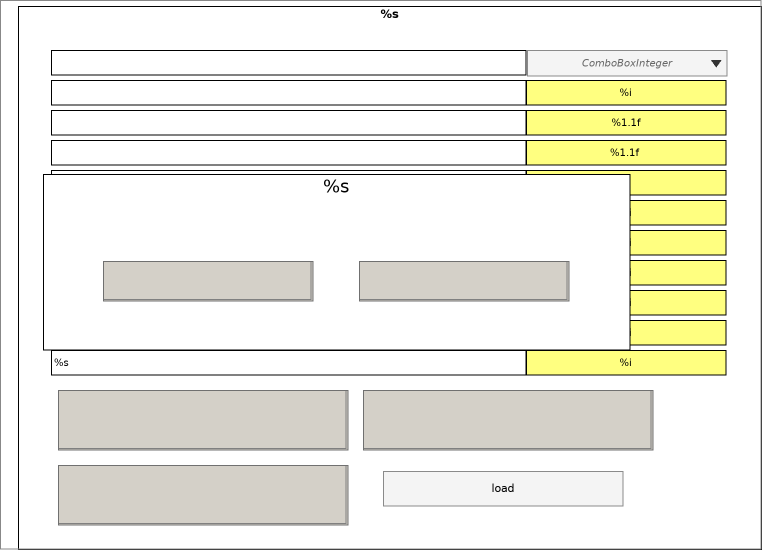
VISUALIZATION VISU_REGENERATION  // 762x550
VAR_IN_OUT
	COM: BLOCK_RS232_ONBOARD_V4;
END_VAR
    RoundedRectangle (18,6 744x544), "%s", text list: 'TextList_CryoPump', text index: 98
    Rectangle (51,50 475x25), text list: 'TextList_CryoPump', text index: 45
    Rectangle (526,140 200x25), "%1.1f", text variable: COM.PRM_PumpRestartDelay, input disabled if: NOT Global_Variables.PRG_USER.ACTU_USER.CONF_MACHINE
        OnMouseClick: write COM.PRM_PumpRestartDelay via Edit
    Rectangle (51,110 475x25), text list: 'TextList_CryoPump', text index: 57
    Rectangle (51,140 475x25), text list: 'TextList_CryoPump', text index: 11
    Rectangle (51,170 475x25), text list: 'TextList_CryoPump', text index: 10
    Rectangle (51,200 475x25), text list: 'TextList_CryoPump', text index: 12
    Rectangle (51,230 475x25), text list: 'TextList_CryoPump', text index: 13
    Rectangle (51,260 475x25), text list: 'TextList_CryoPump', text index: 30
    Progressbar (383,471 240x35), "load", variable: COM.iCounter_Regen_lecture, invisible if: not(COM.VAR_Mem_CO_Lecture)
    Rectangle (526,110 200x25), "%1.1f", text variable: COM.PRM_PumpStartDelay, input disabled if: NOT Global_Variables.PRG_USER.ACTU_USER.CONF_MACHINE
        OnMouseClick: write COM.PRM_PumpStartDelay via Edit
    ComboBoxInteger (527,50 200x26), variable: COM.ID_COMBOBOX, input disabled if: NOT Global_Variables.PRG_USER.ACTU_USER.CONF_MACHINE, text list: 'TextList_CryoPump'
    Rectangle (526,170 200x25), "%i", text variable: COM.PRM_ExtendedPurgeTime, input disabled if: NOT Global_Variables.PRG_USER.ACTU_USER.CONF_MACHINE
        OnMouseClick: write COM.PRM_ExtendedPurgeTime via Edit
    Rectangle (526,200 200x25), "%i", text variable: COM.PRM_RepurgeCycles, input disabled if: NOT Global_Variables.PRG_USER.ACTU_USER.CONF_MACHINE
        OnMouseClick: write COM.PRM_RepurgeCycles via Edit
    Rectangle (526,230 200x25), "%i", text variable: COM.PRM_RepurgeTime, input disabled if: NOT Global_Variables.PRG_USER.ACTU_USER.CONF_MACHINE
        OnMouseClick: write COM.PRM_RepurgeTime via Edit
    Rectangle (526,260 200x25), "%i", text variable: COM.PRM_ROR, input disabled if: NOT Global_Variables.PRG_USER.ACTU_USER.CONF_MACHINE
        OnMouseClick: write COM.PRM_ROR via Edit
    Rectangle (51,290 475x25), text list: 'TextList_CryoPump', text index: 14
    Rectangle (526,290 200x25), "%i", text variable: COM.PRM_RORCycles, input disabled if: NOT Global_Variables.PRG_USER.ACTU_USER.CONF_MACHINE
        OnMouseClick: write COM.PRM_RORCycles via Edit
    Rectangle (51,320 475x25), text list: 'TextList_CryoPump', text index: 29
    Rectangle (526,320 200x25), "%i", text variable: COM.PRM_RoughToPressure, input disabled if: NOT Global_Variables.PRG_USER.ACTU_USER.CONF_MACHINE
        OnMouseClick: write COM.PRM_RoughToPressure via Edit
    Rectangle (51,80 475x25), text list: 'TextList_CryoPump', text index: 17
    Rectangle (526,80 200x25), "%i", text variable: COM.PRM_StartUpTemperature, input disabled if: NOT Global_Variables.PRG_USER.ACTU_USER.CONF_MACHINE
        OnMouseClick: write COM.PRM_StartUpTemperature via Edit
    Progressbar (383,471 240x35), "load", variable: COM.iCounter_Regen_ecriture, invisible if: not(COM.VAR_Mem_CO_Ecriture)
    Button (58,390 290x60), text list: 'TextList_CryoPump', text index: 18
        OnMouseDown: toggle COM.CO_Lecture
    Button (363,390 290x60), input disabled if: NOT Global_Variables.PRG_USER.ACTU_USER.CONF_MACHINE, text list: 'TextList_CryoPump', text index: 19
        OnMouseDown: toggle COM.CO_Ecriture
        OnMouseUp: execute { COM.CO_Ecriture:= false; }
    Button (58,465 290x60), input disabled if: NOT Global_Variables.PRG_USER.ACTU_USER.CONF_MACHINE, text list: 'TextList_CryoPump', text index: 36
        OnMouseDown: execute { COM.Message_confirm_invisible_regen:=false; }
    Rectangle (51,350 475x25), "%s", text list: 'TextList_CryoPump', text index: 96
    Rectangle (526,350 200x25), "%i", text variable: COM.PRM_1st_stage_control_temp, input disabled if: NOT Global_Variables.PRG_USER.ACTU_USER.CONF_MACHINE OR NOT Global_Variables.PRG_USER.MANUFACTURER
        OnMouseClick: write COM.PRM_1st_stage_control_temp via Edit
    Group (43,174 692x182), invisible if: COM.Message_confirm_invisible_regen
        Rectangle (0,0 587x176), "%s", text list: 'TextList_CryoPump', text index: 91
        Button (316,87 210x40), text list: 'TextList_CryoPump', text index: 93
            OnMouseDown: execute { COM.Message_confirm_invisible_regen:=true; }
        Button (60,87 210x40), text list: 'TextList_CryoPump', text index: 92
            OnMouseDown: execute { COM.CO_Param_ParDefaut:=TRUE; }
            OnMouseUp: execute { COM.CO_Param_ParDefaut:= false; }
            OnMouseUp: execute { COM.Message_confirm_invisible_regen:=true; }
END_VISUALIZATION

(* stored: Version 1.1.0.1, ProductVersion 3.1.4026.18
   Visu VISU_REGENERATION: Id {7ad1d399-dee5-49c8-9def-94f749c0dff9} *)
